{attribute 'GeneratedUsingTerminal: EP2001-1000-0016'}
{attribute addProperty BoxType "EP2001-1000-0016"}
{attribute addProperty Description "EP2001-1000 8 Ch. Dig. Output 24V, 0,5A, M8"}
{attribute addProperty Physics "YY"}
{attribute addProperty Id "Group_0AT %Q*Group_99EF3D304Group_1AT %Q*Group_8FCDB3954WcStateAT %I*WcState_0B2B16F91InfoDataAT %I*InfoData_6F19DB2B2"}
{attribute addProperty CRC "3258791590"}
{attribute addProperty Size "11"}
TYPE EP2001_C23D36A6 EXTENDS EtcSlaveBoxBase_77A0E4A7 :
STRUCT
	{attribute addProperty Name "Group_0"}
	Group_0 : Group_99EF3D30;
	{attribute addProperty Name "Group_1"}
	Group_1 : Group_8FCDB395;
	{attribute addProperty Name "WcState"}
	WcState : WcState_0B2B16F9;
	{attribute addProperty Name "InfoData"}
	InfoData : InfoData_6F19DB2B;
END_STRUCT
END_TYPE

(* stored: Version 1.2.0.0, ProductVersion 3.1.4024.11
   DUT EP2001_C23D36A6: Id {ee9b4e29-11a8-4c76-b1dd-4a2bc4a5ba08} *)
